// TIA Portal V18 export
// export: Created 2026-06-12T02:00:00Z, ExportSetting WithDefaults
VAR_GLOBAL   // PLC tag table "PLC_AI_B4_Tags"
   AI_B4_Daq_C AT %MD200 : Real;   // COUNT 0-100
   AI_B4_TPH_Total AT %MD204 : Real;   // FLOW 100-200 T/h
   AI_B4_KG_CM_Main AT %MD208 : Real;   // PRESSURE 7-8 kg/cm2
   AI_B4_DRM_LVL1 AT %MD212 : Real;   // LEVEL 30-80 %
   AI_B4_DRM_LVL2 AT %MD216 : Real;   // LEVEL 30-80 %
   AI_B4_MW_Output AT %MD220 : Real;   // COUNT 0-50 MW
   AI_B4_KG_CM_2 AT %MD224 : Real;   // PRESSURE 7-8 kg/cm2
   AI_B4_Hc_Value AT %MD228 : Real;   // COUNT 0-100
   AI_B4_Temp_AirHeater_In1 AT %MD232 : Real;   // TEMP 50-80 °C
   AI_B4_Temp_AirHeater_In2 AT %MD236 : Real;   // TEMP 50-80 °C
   AI_B4_Temp_AirHeater_In3 AT %MD240 : Real;   // TEMP 50-80 °C
   AI_B4_Temp_AirHeater_Out1 AT %MD244 : Real;   // TEMP 50-80 °C
   AI_B4_Temp_AirHeater_Out2 AT %MD248 : Real;   // TEMP 50-80 °C
   AI_B4_Pres_AH_mmWC_1 AT %MD252 : Real;   // PRESSURE 7-8 mmWC
   AI_B4_Pres_AH_mmWC_2 AT %MD256 : Real;   // PRESSURE 7-8 mmWC
   AI_B4_Pres_AH_Pct_1 AT %MD260 : Real;   // PERCENT 20-80 %
   AI_B4_Temp_AH_Out3 AT %MD264 : Real;   // TEMP 50-80 °C
   AI_B4_Pres_FDH_mmWC AT %MD268 : Real;   // PRESSURE 7-8 mmWC
   AI_B4_RPM_PAF1 AT %MD272 : Real;   // RPM 800-1200 RPM
   AI_B4_Pct_RPC308_SP AT %MD276 : Real;   // PERCENT 20-80 %
   AI_B4_Pct_RPC308_PV AT %MD280 : Real;   // PERCENT 20-80 %
   AI_B4_Pres_PAF1_mmWC AT %MD284 : Real;   // PRESSURE 7-8 mmWC
   AI_B4_Pct_FDF1_SP AT %MD288 : Real;   // PERCENT 20-80 %
   AI_B4_Pct_FDF1_PV AT %MD292 : Real;   // PERCENT 20-80 %
   AI_B4_Pct_FDF1_OUT AT %MD296 : Real;   // PERCENT 20-80 %
   AI_B4_RPM_FDF1 AT %MD300 : Real;   // RPM 800-1200 RPM
   AI_B4_Pct_RPC301_SP AT %MD304 : Real;   // PERCENT 20-80 %
   AI_B4_Pct_RPC301_PV AT %MD308 : Real;   // PERCENT 20-80 %
   AI_B4_Pct_RPC301_OUT AT %MD312 : Real;   // PERCENT 20-80 %
   AI_B4_mA_ESP1 AT %MD316 : Real;   // CURRENT 50-200 mA
   AI_B4_mA_ESP2 AT %MD320 : Real;   // CURRENT 50-200 mA
   AI_B4_mA_ESP3 AT %MD324 : Real;   // CURRENT 50-200 mA
   AI_B4_mA_ESP4 AT %MD328 : Real;   // CURRENT 50-200 mA
   AI_B4_V_ESP1 AT %MD332 : Real;   // COUNT 0-400 V
   AI_B4_V_ESP2 AT %MD336 : Real;   // COUNT 0-400 V
   AI_B4_V_ESP3 AT %MD340 : Real;   // COUNT 0-400 V
   AI_B4_V_ESP4 AT %MD344 : Real;   // COUNT 0-400 V
   AI_B4_Pct_RPC305_SP AT %MD348 : Real;   // PERCENT 20-80 %
   AI_B4_Pct_RPC305_PV AT %MD352 : Real;   // PERCENT 20-80 %
   AI_B4_RPM_IDF1 AT %MD356 : Real;   // RPM 800-1200 RPM
   AI_B4_Pct_RPC305_VFD AT %MD360 : Real;   // PERCENT 20-80 %
   AI_B4_Pct_FDF2_SP AT %MD364 : Real;   // PERCENT 20-80 %
   AI_B4_Pct_FDF2_PV AT %MD368 : Real;   // PERCENT 20-80 %
   AI_B4_Pct_FDF2_OUT AT %MD372 : Real;   // PERCENT 20-80 %
   AI_B4_RPM_FDF2 AT %MD376 : Real;   // RPM 800-1200 RPM
   AI_B4_Pct_RPC306_SP AT %MD380 : Real;   // PERCENT 20-80 %
   AI_B4_Pct_RPC306_PV AT %MD384 : Real;   // PERCENT 20-80 %
   AI_B4_Pct_RPC306_OUT AT %MD388 : Real;   // PERCENT 20-80 %
   AI_B4_RPM_IDF2 AT %MD392 : Real;   // RPM 800-1200 RPM
   AI_B4_Pct_RPC306_VFD AT %MD396 : Real;   // PERCENT 20-80 %
   AI_B4_Pres_FDF_mmWC AT %MD400 : Real;   // PRESSURE 7-8 mmWC
   AI_B4_TEST1_Value AT %MD404 : Real;   // COUNT 0-100
   AI_B4_Pct_PAF1_SP AT %MD408 : Real;   // PERCENT 20-80 %
   AI_B4_Pct_PAF1_PV AT %MD412 : Real;   // PERCENT 20-80 %
   AI_B4_Pres_PAF2_mmWC AT %MD416 : Real;   // PRESSURE 7-8 mmWC
   AI_B4_RPM_PAF2 AT %MD420 : Real;   // RPM 800-1200 RPM
   AI_B4_Pct_RPC308b_SP AT %MD424 : Real;   // PERCENT 20-80 %
   AI_B4_Pct_RPC308b_PV AT %MD428 : Real;   // PERCENT 20-80 %
   AI_B4_Pct_DAM303B_SP AT %MD432 : Real;   // PERCENT 20-80 %
   AI_B4_Pct_DAM304B_SP AT %MD436 : Real;   // PERCENT 20-80 %
END_VAR
